(* CoDeSys 2.3 export: 4545.EXP *)

(* POU hghgh, LD *)
PROGRAM hghgh
VAR
	b1: BOOL;
	k1: BOOL;
	bs: BOOL;
END_VAR
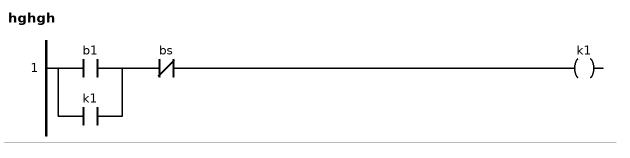
_LD_ (* Ladder Diagram *)
NETWORK 1
	{ [b1] | [k1] } - [/bs] --- (k1)
_END_LD_
(* the same logic as Structured Text *)
(* Network 1 *)
k1 := (b1 OR k1) AND NOT bs;
END_PROGRAM
